Staubli VAL3: onF7Event.pgx

program onF7Event(string x_sId (dimensions=1), bool x_bSave (dimensions=1))
  local string l_sName
  local num i
  local num l_nResult
  local bool l_bFound
  local string l_sButton[2]
  local string l_sMessage
  local bool l_bYes
begin
  // look if the bButton is enable
  if bButton[6]
    //
    // DELETE
    //
    if sMode=="IN" and find(sEvent,"usr")==-1 and find(sEvent,"fast")==-1
      // compose the search "IN,l_sName"
      call alreadyExist(x_sId,l_bFound)
      // if not found
      if !l_bFound
        call language:message(l_sMessage,22)
        // get the yes_no button Key
        call language:getYesNo(l_sButton)
        // ask the question
        call use:yes_no(l_sMessage+sEvent,l_sButton,l_bYes)
        if l_bYes
          call in:setActive(false,x_sId)
          logMsg("[KERNEL] INTERFACE:Disable the Input: "+l_sName)
          x_bSave=true
        endIf
      endIf
    elseIf sMode=="OUT" and find(sEvent,"valve")==-1 and find(sEvent,"fast")==-1
      call alreadyExist(x_sId,l_bFound)
      // if not found
      if !l_bFound
        call language:message(l_sMessage,22)
        // get the yes_no button Key
        call language:getYesNo(l_sButton)
        // ask the question
        call use:yes_no(l_sMessage+sEvent,l_sButton,l_bYes)
        if l_bYes
          call out:setActive(false,x_sId)
          logMsg("[KERNEL] INTERFACE:Disable the Output: "+l_sName)
          x_bSave=true
        endIf
      endIf
    endIf
    // scan the system
    if l_nResult!=0
      // show that the item already exist
      call showExist(l_sName,sMessage)
    endIf
  endIf
end
